(* CoDeSys 2.3 export: STRVALVESTATE.EXP *)

(* Data type *)
(*Состояние 3-х ходового клапана*)
TYPE strValveState :
STRUCT
	Open : BOOL;
	Close: BOOL;
END_STRUCT
END_TYPE
